Staubli VAL3: remMovPoint.pgx

program remMovPoint(trsf& trXYZ[] (dimensions=1), string& sReturn[] (dimensions=1))
  local point pDest
begin
  // Given coordinates, construct the point object for
  // remMoveBase in current frame of reference
  //
  logMsg("call remMovPoint")
  if nIPNumber==0
    pDest=compose(pIP1NullPoint,fIP1,trXYZ)
  else
    pDest=compose(pIP2NullPoint,fIP2,trXYZ)
  endIf
  call remMovBase(pDest,sReturn)
end
